Yaskawa INFORM job: 180_90.JBI

/JOB
//NAME 180_90
///FOLDERNAME OBROTNIK
//POS
///NPOS 0,0,1,0,0,0
///TOOL 0
///POSTYPE PULSE
///PULSE
EC00000=1596314,556476
//INST
///DATE 2025/04/30 12:15
///ATTR SC,RW,RJ
////FRAME ROBOT
///GROUP1 ST1
NOP
MOVJ EC00000 VJ=100.00
END
